// TIA Portal V20 export
// export: Created 2025-12-01T14:56:14.178293Z, ExportSetting None, DisplayName Totally Integrated Automation Portal, DisplayVersion V20 Update 3, DisplayName TIA Portal Openness, DisplayVersion V20 Update 3, DisplayName TIA Portal Version Control Interface, DisplayVersion V20 Update 3, DisplayName STEP 7 Professional, DisplayVersion V20 Update 3, DisplayName STEP 7 Safety, DisplayVersion V20 Update 2, DisplayName WinCC Basic/Comfort/Advanced, DisplayVersion V20 Update 3, DisplayName WinCC Professional, DisplayVersion V20 Update 3, DisplayName WinCC Unified, DisplayVersion V20 Update 3
TYPE "UDT_UTs_Datos"
   STRUCT
      GaliboAltura : USInt;   // Galibo --> Altura
      GaliboAnchura : USInt;   // Galibo --> Anchura
      GaliboProfundidad : USInt;   // Galibo --> Profuncidad
      GaliboTaco : USInt;   // Galibo --> Taco
      GaliboHueco : USInt;   // Galibo --> Hueco
      GaliboHuecoRemontado : USInt;   // Galibo --> Hueco Remontada
      GaliboColor : USInt;   // Galibo --> Color
      GaliboPatin : USInt;   // Galibo --> Patin
      GaliboTipoCarga : USInt;   // Galibo --> Tipo de Carga (Euro,Caja...)
      GaliboRemontada : USInt;   // Galibo --> Carga remontada
      GaliboVacia : USInt;   // Galibo --> Carga Vacia
      CotaAltura : UInt;   // Cota de Altura de la UT
      CotaAnchura : UInt;   // Cota de Anchura de la UT
      CotaProfundidad : UInt;   // Cota de Profundidad de la UT
      Peso : UDInt;   // Peso de la UT
      Presion : USInt;   // Presion para paletizado o despatizado Auto --> Cajas de Plastico
      Amarre : UInt;   // Amarre de la Caja de Palastico
      CodigoEtiquetado : USInt;   // Codigo de Etiquetado de la Carga
      CodigoEnfardado : USInt;   // Codigo de Enfardado de la Carga
      CodigoFlejado : USInt;   // Codigo de Flejado de la Carga
   END_STRUCT;
END_TYPE
